{attribute 'linkalways'} 
{attribute 'no_explicit_call' := 'This FB is a CLASS and must be accessed using methods or properties'}
{attribute 'enable_dynamic_creation'}
FUNCTION_BLOCK FINAL NOT_SINT EXTENDS Node
VAR
	in : _SINT(0);
	out : _SINT(0);
END_VAR

METHOD PUBLIC Clone : I_Node
VAR
	pNode : POINTER TO NOT_SINT;
END_VAR
pNode := __NEW(NOT_SINT);
Clone := pNode^;
END_METHOD

METHOD FB_init : BOOL
VAR_INPUT
	bInitRetains : BOOL; // if TRUE, the retain variables are initialized (warm start / cold start)
	bInCopyCode : BOOL;  // if TRUE, the instance afterwards gets moved into the copy code (online change)
END_VAR
AddInput('in',THIS^.in);
AddOutput('out', THIS^.out);
END_METHOD

METHOD PROTECTED OnExecute
VAR
END_VAR
out.Value := NOT in.Value;
END_METHOD

END_FUNCTION_BLOCK

(* stored: Version 1.1.0.1, ProductVersion 3.1.4024.15
   POU NOT_SINT: Id {0d69c1e3-77c2-4a26-8988-82fe95309aed}, SpecialFunc None
   Folder Constructor: Id {c130eecf-a34b-459b-b820-4f1af99e9d35}
   Method Clone: Id {46c04801-7e4b-475a-96a7-7ad358bba3cb}
   Method FB_init: Id {6f4e6838-6009-40f4-917a-99bd88992cb1}
   Method OnExecute: Id {17b5e87b-960e-46ab-a173-7b619f0833d6} *)
